FUNCTION_BLOCK FB_LamparaComputada_IL
// La lampara se enciende tras un determinado numero de pulsaciones
// La lampara se apaga tras accionar el pulsador de reinicio
VAR_INPUT
    ManiobrasTotales     : UINT := 2;
END_VAR
VAR_OUTPUT
    ManiobrasPendientes  : UINT;
END_VAR
VAR
    Contador                  : CTD := (CV := ManiobrasTotales);
    Lampara           AT %Q*  : BOOL;
    Pulsador          AT %I*  : BOOL;
    PulsadorReinicio  AT %I*  : BOOL;
END_VAR

// NETWORK 1
// instruction list
CAL     Contador(
    CD      := Pulsador,
    LOAD    := PulsadorReinicio,
    PV      := ManiobrasTotales)

// NETWORK 2
// instruction list
LD      Contador.Q
ST      Lampara

// NETWORK 3
// instruction list
LD      Contador.CV
ST      ManiobrasPendientes

END_FUNCTION_BLOCK

(* stored: Version 1.1.0.1, ProductVersion 3.1.4024.15
   POU FB_LamparaComputada_IL: Id {93535b98-fe33-48e8-8ef0-b43c79734c24}, SpecialFunc None *)
